// Mitsubishi GX Works2 project: PULSE X0   PLC: Q03UDV

PROGRAM MAIN
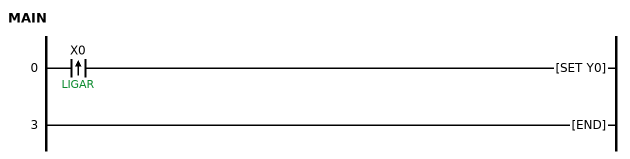
0     LDP     X0  ; LIGAR
      SET     Y0
3     END
END_PROGRAM

// device comments not shown above
X1  ; DESLIGAR
